PROGRAM PRG_11_AirFlowAnalytics
VAR
	AirFlowRateSensor: GenericSensor;
	AirPressureSensor: GenericSensor;
	AirTemperatureSensor: GenericSensor;
	
	AirFlowSensorPostHttp: HttpPost;
	AirPresSensorPostHttp: HttpPost;
	AirTempSensorPostHttp: HttpPost;
END_VAR

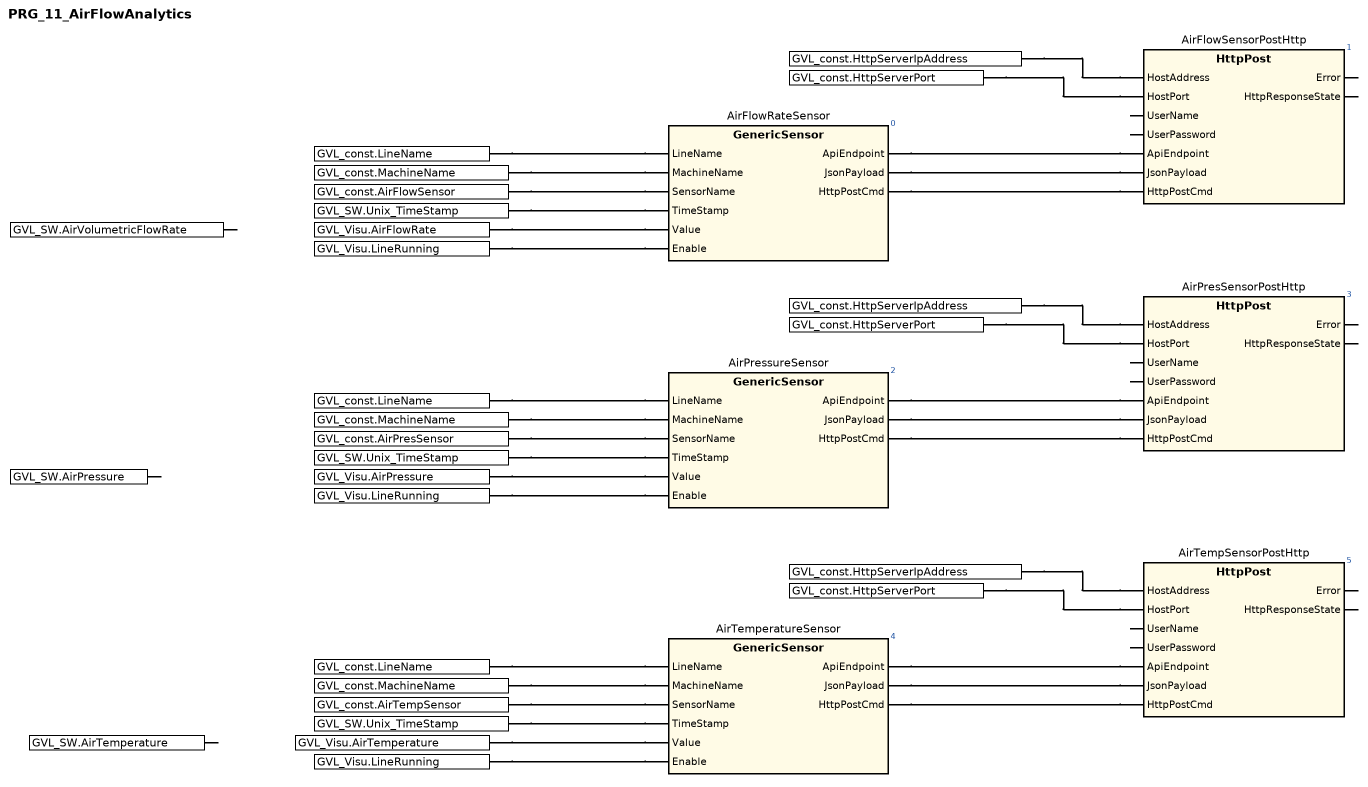
AirFlowRateSensor(
    LineName := GVL_const.LineName,
    MachineName := GVL_const.MachineName,
    SensorName := GVL_const.AirFlowSensor,
    TimeStamp := GVL_SW.Unix_TimeStamp,
    Value := GVL_Visu.AirFlowRate,
    Enable := GVL_Visu.LineRunning); // GenericSensor
AirFlowSensorPostHttp(
    HostAddress := GVL_const.HttpServerIpAddress,
    HostPort := GVL_const.HttpServerPort,
    ApiEndpoint := AirFlowRateSensor.ApiEndpoint,
    JsonPayload := AirFlowRateSensor.JsonPayload,
    HttpPostCmd := AirFlowRateSensor.HttpPostCmd); // HttpPost
AirPressureSensor(
    LineName := GVL_const.LineName,
    MachineName := GVL_const.MachineName,
    SensorName := GVL_const.AirPresSensor,
    TimeStamp := GVL_SW.Unix_TimeStamp,
    Value := GVL_Visu.AirPressure,
    Enable := GVL_Visu.LineRunning); // GenericSensor
AirPresSensorPostHttp(
    HostAddress := GVL_const.HttpServerIpAddress,
    HostPort := GVL_const.HttpServerPort,
    ApiEndpoint := AirPressureSensor.ApiEndpoint,
    JsonPayload := AirPressureSensor.JsonPayload,
    HttpPostCmd := AirPressureSensor.HttpPostCmd); // HttpPost
AirTemperatureSensor(
    LineName := GVL_const.LineName,
    MachineName := GVL_const.MachineName,
    SensorName := GVL_const.AirTempSensor,
    TimeStamp := GVL_SW.Unix_TimeStamp,
    Value := GVL_Visu.AirTemperature,
    Enable := GVL_Visu.LineRunning); // GenericSensor
AirTempSensorPostHttp(
    HostAddress := GVL_const.HttpServerIpAddress,
    HostPort := GVL_const.HttpServerPort,
    ApiEndpoint := AirTemperatureSensor.ApiEndpoint,
    JsonPayload := AirTemperatureSensor.JsonPayload,
    HttpPostCmd := AirTemperatureSensor.HttpPostCmd); // HttpPost
// GVL_SW.AirVolumetricFlowRate: input not connected
// GVL_SW.AirPressure: input not connected
// GVL_SW.AirTemperature: input not connected

END_PROGRAM

(* stored: Version 1.1.0.1, ProductVersion 3.1.4024.15
   POU PRG_11_AirFlowAnalytics: Id {96d35d53-1242-4be7-b36c-7cd64f603641}, SpecialFunc None *)
